{attribute 'linkalways'} 
{attribute 'no_explicit_call' := 'This FB is a CLASS and must be accessed using methods or properties'}
{attribute 'enable_dynamic_creation'}
FUNCTION_BLOCK FINAL GE_DWORD EXTENDS Node
VAR
	in1 : _DWORD(0);
	in2 : _DWORD(0);
	out : _BOOL(FALSE);
END_VAR

METHOD PUBLIC Clone : I_Node
VAR
	pNode : POINTER TO GE_DWORD;
END_VAR
pNode := __NEW(GE_DWORD);
Clone := pNode^;
END_METHOD

METHOD FB_init : BOOL
VAR_INPUT
	bInitRetains : BOOL; // if TRUE, the retain variables are initialized (warm start / cold start)
	bInCopyCode : BOOL;  // if TRUE, the instance afterwards gets moved into the copy code (online change)
END_VAR
AddInput('in1',THIS^.in1);
AddInput('in2',THIS^.in2);
AddOutput('out', THIS^.out);
END_METHOD

METHOD PROTECTED OnExecute
VAR
END_VAR
out.Value := in1.Value >= in2.Value;
END_METHOD

END_FUNCTION_BLOCK

(* stored: Version 1.1.0.1, ProductVersion 3.1.4024.15
   POU GE_DWORD: Id {5b01f21f-2cb6-41d7-b86f-73c3e5f23713}, SpecialFunc None
   Folder Constructor: Id {63e7a055-fc32-40c9-a31a-a4f9300e2170}
   Method Clone: Id {427d4120-cce2-44b8-bc46-aff593359c5f}
   Method FB_init: Id {08a974c5-ac79-4405-b906-23e5a5856c56}
   Method OnExecute: Id {f78adcfc-d22c-4440-afcb-3ae3c5ad1579} *)
